FUNCTION_BLOCK Part IMPLEMENTS IPart
VAR_INPUT
END_VAR
VAR_OUTPUT
END_VAR
VAR
	_id: STRING(23);
END_VAR

{warning 'Eigenschaftenimplementierung hinzufügen'}
PROPERTY id : STRING(23)
GET
id := THIS^._id;
END_GET
SET
THIS^._id := id;
END_SET
END_PROPERTY

END_FUNCTION_BLOCK

(* stored: Version 1.1.0.1
   POU Part: Id {145af6aa-7eef-4f55-81b6-6669a433a0e0}, SpecialFunc None
   Property id: Id {4860a955-db7d-453f-8591-8ce619d56edf}
   Get Get: Id {9111c330-3dfa-481a-95c2-1003863ff486}
   Set Set: Id {90b7afc8-23b0-42a6-b0b4-b07adcc8716c} *)
